# EPICS StreamDevice protocol: pdsgo2/Db/pdsgo2.proto
# pdsgo2.proto

InTerminator = LF CR;
OutTerminator = LF;

ReplyTimeout = 2000;
#ReadTimeout = 500;

get_data {
   out "#gw";
   in "#Rw, %d,%(\$1)d,%(\$2)d,%(\$3)d,%(\$4)d,%(\$5.RVAL)f, %(\$6.RVAL)f,%(\$7)i";
   @mismatch {
       in "%(\$8)s";
   }
}
